FUNCTION_BLOCK SP_Stoppering (* Stoppering parameters (none): OPC UA IDs, range check and latching *)
  (* Standard: 61499-2 *)
  (* Version 0.1, 2026-09-28, Project contributors, AAU Smart Production Lab *)
  PACKAGE stoppering;
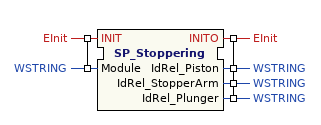
  EVENT_INPUT
    INIT : EInit WITH Module;
  END_EVENT
  EVENT_OUTPUT
    INITO : EInit WITH IdRel_Piston, IdRel_StopperArm, IdRel_Plunger;
  END_EVENT
  VAR_INPUT
    Module : WSTRING;
  END_VAR
  VAR_OUTPUT
    IdRel_Piston : WSTRING;
    IdRel_StopperArm : WSTRING;
    IdRel_Plunger : WSTRING;
  END_VAR
  EC_STATES
    INIT : INIT -> INITO;
  END_STATES
  ALGORITHM INIT IN ST:
IdRel_Piston := CONCAT(CONCAT("loc[", Module), "/Piston/cmd]");
IdRel_StopperArm := CONCAT(CONCAT("loc[", Module), "/StopperArm/cmd]");
IdRel_Plunger := CONCAT(CONCAT("loc[", Module), "/Plunger/cmd]");
  END_ALGORITHM
END_FUNCTION_BLOCK
